// TwinCAT 3 PLC project ClientSampleProject
// ProgramVersion: 3.1.0.8
// libraries:
//   Tc2_Standard, * (Beckhoff Automation GmbH)
//   Tc2_System, * (Beckhoff Automation GmbH)
//   Tc3_Interfaces, * (Beckhoff Automation GmbH)
//   Tc3_Module, * (Beckhoff Automation GmbH)
//   Tc3_PLCopen_OpcUa, * (Beckhoff Automation GmbH)
//   Tc2_Utilities,newest,Beckhoff Automation GmbH
// project tree:
//   DUTs/ ST_OutputArgInfoAndData.TcDUT, ST_ReadListData.TcDUT (not stored), ST_ReadListData_Array.TcDUT
//   GVLs/ GlobalSettings.TcGVL
//   / PlcTask.TcTTO (not stored)
//   POUs/ MAIN.TcPOU, PRG_METHOD.TcPOU, PRG_READ.TcPOU, PRG_READ_IndexRange.TcPOU, PRG_READ_List.TcPOU, PRG_READ_List_Array.TcPOU, PRG_WRITE.TcPOU, PRG_WRITE_IndexRange.TcPOU
// (motion and I/O tree: see PLC project serversampleproject)
// real-time tasks:
//   TASK PlcTask: cycle T#10ms, priority 20, ADS port 350

// ---- DUTs/ST_OutputArgInfoAndData.TcDUT
{attribute 'pack_mode' := '1'}
TYPE ST_OutputArgInfoAndData :
STRUCT
	nNumberOfOutputArguments: UDINT; // determined amount of output parameters
	nReserved: ARRAY[1..4] OF BYTE; // Reserved padding
	stOutputArgInfo: ARRAY[1..1] OF ST_UAMethodArgInfo; // number of output parameters - M_Mul has 1 output parameter 
	pro: DINT;
END_STRUCT
END_TYPE

// ---- DUTs/ST_ReadListData_Array.TcDUT
{attribute 'pack_mode' := '1'}
TYPE ST_ReadListData_Array :
STRUCT
	stReadListReturnInfo	: ARRAY [1..2] OF ST_UAReadListReturnInfo;
	iArrayIntVar1 			: ARRAY[0..9] OF INT;
	iArrayIntVar2 			: ARRAY[0..11] OF INT;
END_STRUCT
END_TYPE

// ---- GVLs/GlobalSettings.TcGVL
VAR_GLOBAL
	(* These global connection and namespace settings need to be adapted to the runtime environment *)
	(*sOpcUaServerUrl : STRING(MAX_STRING_LENGTH) := 'opc.tcp://localhost:4840';
	sNamespaceUri : STRING(MAX_STRING_LENGTH) := 'urn:BeckhoffAutomation:Ua:PLC1'; // TF6100 setup version 4.x default*)
	
	sOpcUaServerUrl : STRING(MAX_STRING_LENGTH) := 'opc.tcp://172.17.36.240:4840';
	sNamespaceUri : STRING(MAX_STRING_LENGTH) := 'urn:BeckhoffAutomation:Ua:PLC1'; // TF6100 setup version 4.x default
END_VAR

// ---- POUs/MAIN.TcPOU
PROGRAM MAIN
VAR
	fbGetHostname : FB_GetHostName;
END_VAR

PRG_READ(); // Call sample for UA_Read
//PRG_READ_IndexRange(); // Call sample for UA_Read
//PRG_READ_List(); // Call sample for UA_ReadList
//PRG_READ_List_Array(); // Call sample for UA_ReadList to read array elements
//PRG_WRITE(); // Call sample for UA_Write
//PRG_WRITE_IndexRange(); // Call sample for UA_Write
//PRG_METHOD(); // Call sample for UA_MethodCall

END_PROGRAM

// ---- POUs/PRG_READ.TcPOU
PROGRAM PRG_READ
VAR
	(* Declarations for UA_Connect *)
	fbUA_Connect			: UA_Connect;
	SessionConnectInfo		: ST_UASessionConnectInfo;
	nConnectionHdl			: DWORD;

	(* Declarations for UA_GetNamespaceIndex *)
	fbUA_GetNamespaceIndex 	: UA_GetNamespaceIndex;
	nNamespaceIndex			: UINT;

	(* Declarations for UA_NodeGetHandle *)
	fbUA_NodeGetHandle		: UA_NodeGetHandle;
	NodeID					: ST_UANodeID;
	nNodeHdl				: DWORD;

	(* Declarations for UA_Read *)
	fbUA_Read				: UA_Read;
	stIndexRange			: ARRAY [1..nMaxIndexRange] OF ST_UAIndexRange;
	nIndexRangeCount		: UINT;
	stNodeAddInfo			: ST_UANodeAdditionalInfo;
	sNodeIdentifier			: STRING(MAX_STRING_LENGTH) := 'MAIN.nCounter'; // change to node identifier
	nReadData				: INT; 		// change to node data type
	cbDataRead				: UDINT;
	
	(* Declarations for UA_NodeReleaseHandle *)
	fbUA_NodeReleaseHandle	: UA_NodeReleaseHandle;

	(* Declarations for UA_Disconnect *)
	fbUA_Disconnect		: UA_Disconnect;

	(* Other declarations *)
	iState		: INT;
	bTest		: BOOL:= TRUE;
	bDone		: BOOL;
	bBusy		: BOOL;
	bError		: BOOL;
	nErrorID	: DWORD;
END_VAR


CASE iState OF
0:	(* idle *)
	IF bTest THEN
		bTest		:= FALSE;
		bError		:= FALSE;
		nErrorID	:= 0;

		SessionConnectInfo.tConnectTimeout 		:= T#1M;
		SessionConnectInfo.tSessionTimeout 		:= T#1M;
		SessionConnectInfo.sApplicationName		:= '';
		SessionConnectInfo.eSecurityMode 		:= eUASecurityMsgMode_Sign_Encrypt;
		SessionConnectInfo.eSecurityPolicyUri 	:= 5;
		SessionConnectInfo.eTransportProfileUri := eUATransportProfileUri_UATcp;

(*		nIndexRange[1].nStartIndex := 0;
		nIndexRange[1].nEndIndex := 1;
		nIndexRange[1].bRangeAccess := TRUE; *)
		stNodeAddInfo.nIndexRangeCount := nIndexRangeCount;
		stNodeAddInfo.stIndexRange := stIndexRange;
		iState	:= iState + 1;
	END_IF

1:	(* Open UA session *)
	fbUA_Connect(
		Execute				:= TRUE,
		ServerURL			:= sOpcUaServerUrl,
		SessionConnectInfo	:= SessionConnectInfo,
		Timeout				:= T#2M,
		ConnectionHdl		=> nConnectionHdl
	);

	IF NOT fbUA_Connect.Busy THEN
		fbUA_Connect(Execute := FALSE);

		IF NOT fbUA_Connect.Error THEN
			(* session open *)
			iState := iState + 1;
		ELSE
			bError			:= TRUE;
			nErrorID		:= fbUA_Connect.ErrorID;
			nConnectionHdl	:= 0;
			iState 			:= 0; (* idle *)
		END_IF
	END_IF


2:	(* GetNS Index *)
	fbUA_GetNamespaceIndex(
		Execute			:= TRUE,
		ConnectionHdl	:= nConnectionHdl,
		NamespaceUri	:= sNamespaceUri,
		NamespaceIndex	=> nNamespaceIndex
	);

	IF NOT fbUA_GetNamespaceIndex.Busy THEN
		fbUA_GetNamespaceIndex(Execute := FALSE);
		IF NOT fbUA_GetNamespaceIndex.Error THEN
			iState 		:= iState + 1;
		ELSE
			bError		:= TRUE;
			nErrorID	:= fbUA_GetNamespaceIndex.ErrorID;
			iState 		:= 6; (* idle *)
		END_IF
	END_IF

3:	(* Get Node Handle *)
	NodeID.eIdentifierType := eUAIdentifierType_String;
	NodeID.nNamespaceIndex := nNamespaceIndex;
	NodeID.sIdentifier	:= sNodeIdentifier;
	fbUA_NodeGetHandle(
		Execute			:= TRUE,
		ConnectionHdl	:= nConnectionHdl,
		NodeID			:= NodeID,
		NodeHdl			=> nNodeHdl
	);

	IF NOT fbUA_NodeGetHandle.Busy THEN
		fbUA_NodeGetHandle(Execute := FALSE);

		IF NOT fbUA_NodeGetHandle.Error THEN
			iState 		:= iState + 1;
		ELSE
			bError		:= TRUE;
			nErrorID	:= fbUA_NodeGetHandle.ErrorID;
			iState 		:= 6; (* idle *)
		END_IF
	END_IF


4: 	(* UA_Read *)
	fbUA_Read(
		Execute			:= TRUE,
		ConnectionHdl	:= nConnectionHdl,
		NodeHdl			:= nNodeHdl,
		cbData			:= SIZEOF(nReadData),
		stNodeAddInfo 	:= stNodeAddInfo,
		pVariable		:= ADR(nReadData)
		);

	IF NOT fbUA_Read.Busy THEN
		fbUA_Read( Execute := FALSE, cbData_R => cbDataRead);

		IF NOT fbUA_Read.Error THEN
			iState 		:= iState + 1;
		ELSE
			bError		:= TRUE;
			nErrorID	:= fbUA_Read.ErrorID;
			iState 		:= 6; (* idle *)
		END_IF
	END_IF


5:	(* Release Node Handle *)
	fbUA_NodeReleaseHandle(
		Execute			:= TRUE,
		ConnectionHdl	:= nConnectionHdl,
		NodeHdl			:= nNodeHdl
	);

	IF NOT fbUA_NodeReleaseHandle.Busy THEN
		fbUA_NodeReleaseHandle(Execute := FALSE);

		IF NOT fbUA_NodeReleaseHandle.Error THEN
			iState 		:= iState + 1;
		ELSE
			bError		:= TRUE;
			nErrorID	:= fbUA_NodeReleaseHandle.ErrorID;
			iState 		:= 6; (* idle *)
		END_IF
	END_IF


6:	(* close session *)
	fbUA_Disconnect(
		Execute			:= TRUE,
		ConnectionHdl	:= nConnectionHdl
	);

	IF NOT fbUA_Disconnect.Busy THEN
		fbUA_Disconnect(Execute := FALSE);
		bBusy := FALSE;
		IF NOT fbUA_Disconnect.Error THEN
			(* session closed *)
			iState 		:= 0;
			IF NOT bError THEN 
				bDone 	:= TRUE;
			END_IF
		ELSE
			bError			:= TRUE;
			nErrorID		:= fbUA_Disconnect.ErrorID;
			iState 			:= 0; (* idle *)
			nConnectionHdl	:= 0;
		END_IF
	END_IF
END_CASE

END_PROGRAM

// ---- POUs/PRG_METHOD.TcPOU
PROGRAM PRG_METHOD
VAR
	(* Declarations for UA_Connect *)	
	fbUA_Connect: UA_Connect;
	SessionConnectInfo: ST_UASessionConnectInfo;
	nConnectionHdl: DWORD;
	
	(* Declarations for UA_GetNamespaceIndex *)
	fbUA_GetNamespaceIndex: UA_GetNamespaceIndex;
	nNamespaceIndex: UINT;
	
	(* Declarations for UA_MethodGetHandle *)
	fbUA_MethodGetHandle: UA_MethodGetHandle;
	ObjectNodeID: ST_UANodeID;
	MethodNodeID: ST_UANodeID;
	nMethodHdl: DWORD;
	
	(* Declarations for UA_MethodCall *)
	fbUA_MethodCall: UA_MethodCall;
	sObjectNodeIdIdentifier	: STRING(MAX_STRING_LENGTH) := 'MAIN.fbMathematics'; // change to object node identifier (UAObject above method)
	sMethodNodeIdIdentifier : STRING(MAX_STRING_LENGTH) := 'MAIN.fbMathematics#M_Mul'; // change to method node identifier (UAMethod to call)
	nAdrWriteData: PVOID;
	numberIn1: INT := 42; // change according to input value and data type
	numberIn2: INT := 42; // change according to input value and data type
	numberOutPro: DINT; // result (output parameter of M_Mul())
	cbWriteData: UDINT; // calculated automatically by M_Init()
	InputArguments: ARRAY[1..2] OF ST_UAMethodArgInfo; // change according to input parameters - M_Mul has 2 input parameters 
	stOutputArgInfo: ARRAY[1..1] OF ST_UAMethodArgInfo; // change according to output parameters - M_Mul has 1 output parameters
	stOutputArgInfoAndData: ST_OutputArgInfoAndData;
	nInputData: ARRAY[1..4] OF BYTE; // numberIn1(INT16)(2) + numberIn2(INT16)(2)
	nOffset: UDINT; // calculated by M_Init()
	nArg: INT; // used by M_Init()
	
	(* Declarations for UA_MethodReleaseHandle *)
	fbUA_MethodReleaseHandle: UA_MethodReleaseHandle;

	(* Declarations for UA_Disconnect *)
	fbUA_Disconnect: UA_Disconnect;
			
	(* Other Declarations *)
	bTest: BOOL := TRUE;
	bDone: BOOL;
	bBusy: BOOL;
	bError: BOOL;
	nErrorID: DWORD;
	iState: INT;
	RTrig: R_TRIG;
	bInputDataError: BOOL;
END_VAR
VAR CONSTANT
	nInputArgSize: INT := 4; // numberIn1(INT16)(2) + numberIn2(INT16)(2)
	nNumberOfInputArguments: DINT := 2; // change to number of input parameters - M_Mul has 2 input parameters
	nNumberOfOutputArguments: DINT := 1; // change to number of output parameters - M_Mul has 1 output parameters
END_VAR

CASE iState OF

0:	(* idle *)
	IF bTest THEN
		bTest		:= FALSE;
		bError		:= FALSE;
		nErrorID	:= 0;

		SessionConnectInfo.tConnectTimeout 		:= T#1M;
		SessionConnectInfo.tSessionTimeout 		:= T#1M;
		SessionConnectInfo.sApplicationName		:= '';
		SessionConnectInfo.eSecurityMode 		:= eUASecurityMsgMode_None;
		SessionConnectInfo.eSecurityPolicyUri 	:= eUASecurityPolicy_None;
		SessionConnectInfo.eTransportProfileUri := eUATransportProfileUri_UATcp;

		iState	:= iState + 1;
	END_IF

	
1:	(* open UA session *)
	fbUA_Connect(
		Execute				:= TRUE,
		ServerURL			:= sOpcUaServerUrl,
		SessionConnectInfo	:= SessionConnectInfo,
		Timeout				:= T#2M,
		ConnectionHdl		=> nConnectionHdl
	);

	IF NOT fbUA_Connect.Busy THEN
		fbUA_Connect(Execute := FALSE);

		IF NOT fbUA_Connect.Error THEN
			(* connected *)
			iState := iState + 1;
		ELSE
			bError			:= TRUE;
			nErrorID		:= fbUA_Connect.ErrorID;
			nConnectionHdl	:= 0;
			iState 			:= 0; (* idle *)
		END_IF
	END_IF


2:	(* GetNS Index *)
	fbUA_GetNamespaceIndex(
		Execute			:= TRUE,
		ConnectionHdl	:= nConnectionHdl,
		NamespaceUri	:= sNamespaceUri,
		NamespaceIndex	=> nNamespaceIndex
	);

	IF NOT fbUA_GetNamespaceIndex.Busy THEN
		fbUA_GetNamespaceIndex(Execute := FALSE);

		IF NOT fbUA_GetNamespaceIndex.Error THEN
			(* namespace index read successfully *)
			iState 		:= iState + 1;
		ELSE
			bError		:= TRUE;
			nErrorID	:= fbUA_GetNamespaceIndex.ErrorID;
			iState 		:= 7; (* disconnect *)
		END_IF
	END_IF

	
3:	(* Get Method Handle *)
	ObjectNodeID.eIdentifierType := eUAIdentifierType_String;
	ObjectNodeID.nNamespaceIndex := nNamespaceIndex;
	ObjectNodeID.sIdentifier	 := sObjectNodeIdIdentifier;

	MethodNodeID.eIdentifierType := eUAIdentifierType_String;
	MethodNodeID.nNamespaceIndex := nNamespaceIndex;
	MethodNodeID.sIdentifier	 := sMethodNodeIdIdentifier;

	M_Init();
	IF bInputDataError = FALSE THEN
		iState 	:= iState + 1;
	ELSE
		bBusy		:= FALSE;  
		bError 		:= TRUE;
		nErrorID 	:= 16#70A; //out of memory
	END_IF

	
4:	(* Method Get Handle *)
	fbUA_MethodGetHandle(
			Execute			:= TRUE,
			ConnectionHdl	:= nConnectionHdl,
			ObjectNodeID	:= ObjectNodeID,
			MethodNodeID 	:= MethodNodeID,
			MethodHdl		=> nMethodHdl
		);
	IF NOT fbUA_MethodGetHandle.Busy THEN
		fbUA_MethodGetHandle(Execute := FALSE);

		IF NOT fbUA_MethodGetHandle.Error THEN
			(*  *)
			iState := iState + 1; (* Call Method *)
		ELSE
			bError		:= TRUE;
			nErrorID	:= fbUA_MethodGetHandle.ErrorID;
			iState	 	:= 6; (* Release method Handle *)
		END_IF
	END_IF


5:	(* Method Call *)
	stOutputArgInfo[1].nLenData := SIZEOF(stOutputArgInfoAndData.pro);
	fbUA_MethodCall(
		Execute					:= TRUE,
		ConnectionHdl			:= nConnectionHdl,
		MethodHdl				:= nMethodHdl,
		nNumberOfInputArguments := nNumberOfInputArguments,	
		pInputArgInfo			:= ADR(InputArguments),
		cbInputArgInfo			:= SIZEOF(InputArguments),
		pInputArgData			:= ADR(nInputData),
		cbInputArgData			:= cbWriteData,
		pInputWriteData			:= 0,
		cbInputWriteData		:= 0,
		nNumberOfOutputArguments:= nNumberOfOutputArguments,
		pOutputArgInfo			:= ADR(stOutputArgInfo),
		cbOutputArgInfo			:= SIZEOF(stOutputArgInfo),
		pOutputArgInfoAndData	:= ADR(stOutputArgInfoAndData),
		cbOutputArgInfoAndData	:= SIZEOF(stOutputArgInfoAndData),		
	);
	IF NOT fbUA_MethodCall.Busy THEN
		fbUA_MethodCall(Execute := FALSE);
		IF NOT fbUA_MethodCall.Error THEN
			(* clear data and restart *)
			iState := iState + 1; (* Release handle *)
			numberOutPro := stOutputArgInfoAndData.pro;
		ELSE
			bError		:= TRUE;
			nErrorID	:= fbUA_MethodCall.ErrorID;
			iState		:= 6; (* Release method handle *)
		END_IF
	END_IF


6:	(* Release Method Handle *)
	fbUA_MethodReleaseHandle(
		Execute			:= TRUE,
		ConnectionHdl	:= nConnectionHdl,
		MethodHdl		:= nMethodHdl
	);

	IF NOT fbUA_MethodReleaseHandle.Busy THEN
		fbUA_MethodReleaseHandle(Execute := FALSE);
		bBusy := FALSE;
		IF NOT fbUA_MethodReleaseHandle.Error THEN
			(* session closed *)
			iState 	:= 7; (* Disconnect *)
		ELSE
			bError		:= TRUE;
			nErrorID	:= fbUA_MethodReleaseHandle.ErrorID;
			iState 		:= 7; (* Disconnect *)
		END_IF
	END_IF
	
	
7:	(* Disconnect *) 
	fbUA_Disconnect(
		Execute			:= TRUE,
		ConnectionHdl	:= nConnectionHdl
	);

	IF NOT fbUA_Disconnect.Busy THEN
		fbUA_Disconnect(Execute := FALSE);

		IF NOT fbUA_Disconnect.Error THEN
			(* disconnected *)
			iState 	:= 0; (* idle *)
			bDone 	:= TRUE;
			bBusy 	:= FALSE;
		ELSE
			bBusy 			:= FALSE;
			bError			:= TRUE;
			nErrorID		:= fbUA_Disconnect.ErrorID;
			iState 			:= 0; (* idle *)
			nConnectionHdl	:= 0;
		END_IF
	END_IF
END_CASE

ACTION M_Init:
bInputDataError := FALSE; 
nOffset := 0;
MEMSET(ADR(InputArguments),0,SIZEOF(InputArguments));
MEMSET(ADR(nInputData),0,SIZEOF(nInputData));

nArg := 1;
(*numberIn1*)			(********** Input parameter 1 **********)
InputArguments[nArg].DataType			:= eUAType_Int16;
InputArguments[nArg].ValueRank			:= -1; 							(* Scalar = -1 or Array *)
InputArguments[nArg].ArrayDimensions[1]	:= 0; 							(* Number of Dimension in case its an array *)
InputArguments[nArg].nLenData			:= SIZEOF(numberIn1);			(* Length if its a STRING *)
IF nOffset + SIZEOF(numberIn1) > nInputArgSize THEN 
	bInputDataError := TRUE;
	RETURN;
ELSE
	MEMCPY(ADR(nInputData)+nOffset,ADR(numberIn1),SIZEOF(numberIn1));				(* VALUE in BYTES FORM *)
	nOffset := nOffset + SIZEOF(numberIn1);
END_IF

nArg := nArg + 1;
(* numberIn2;*)			(********** Input parameter 2 **********)
InputArguments[nArg].DataType			:= eUAType_Int16;
InputArguments[nArg].ValueRank			:= -1; 							(* Scalar = -1 or Array *)
InputArguments[nArg].ArrayDimensions[1]	:= 0; 							(* Number of Dimension in case its an array *)
InputArguments[nArg].nLenData			:= SIZEOF(numberIn2);				(* Length if its a STRING *)
IF nOffset + SIZEOF(numberIn2) > nInputArgSize THEN 
	bInputDataError := TRUE;
	RETURN;
ELSE
	MEMCPY(ADR(nInputData)+nOffset,ADR(numberIn2),SIZEOF(numberIn2));			(* VALUE in BYTES FORM *)
	nOffset := nOffset + SIZEOF(numberIn2);
END_IF

cbWriteData := nOffset;
END_ACTION

END_PROGRAM

// ---- POUs/PRG_READ_IndexRange.TcPOU
PROGRAM PRG_READ_IndexRange
VAR
	(* Declarations for UA_Connect *)
	fbUA_Connect			: UA_Connect;
	SessionConnectInfo		: ST_UASessionConnectInfo;
	nConnectionHdl			: DWORD;

	(* Declarations for UA_GetNamespaceIndex *)
	fbUA_GetNamespaceIndex 	: UA_GetNamespaceIndex;
	nNamespaceIndex			: UINT;

	(* Declarations for UA_NodeGetHandle *)
	fbUA_NodeGetHandle		: UA_NodeGetHandle;
	NodeID					: ST_UANodeID;
	nNodeHdl				: DWORD;

	(* Declarations for UA_Read *)
	fbUA_Read				: UA_Read;
	stIndexRange			: ARRAY [1..nMaxIndexRange] OF ST_UAIndexRange;
	//nIndexRangeCount		: UINT;
	stNodeAddInfo			: ST_UANodeAdditionalInfo;
	sNodeIdentifier			: STRING(MAX_STRING_LENGTH) := 'MAIN.iArrayIntVar3'; // change to node identifier
	nReadData				: ARRAY[0..3] OF DINT; 		// change to node data type
	cbDataRead				: UDINT;
	
	(* Declarations for UA_NodeReleaseHandle *)
	fbUA_NodeReleaseHandle	: UA_NodeReleaseHandle;

	(* Declarations for UA_Disconnect *)
	fbUA_Disconnect		: UA_Disconnect;

	(* Other declarations *)
	iState		: INT;
	bTest		: BOOL:= TRUE;
	bDone		: BOOL;
	bBusy		: BOOL;
	bError		: BOOL;
	nErrorID	: DWORD;
END_VAR


CASE iState OF
0:	(* idle *)
	IF bTest THEN
		bTest		:= FALSE;
		bError		:= FALSE;
		nErrorID	:= 0;

		SessionConnectInfo.tConnectTimeout 		:= T#1M;
		SessionConnectInfo.tSessionTimeout 		:= T#1M;
		SessionConnectInfo.sApplicationName		:= '';
		SessionConnectInfo.eSecurityMode 		:= eUASecurityMsgMode_None;
		SessionConnectInfo.eSecurityPolicyUri 	:= eUASecurityPolicy_None;
		SessionConnectInfo.eTransportProfileUri := eUATransportProfileUri_UATcp;

		stIndexRange[1].nStartIndex := 2;
		stIndexRange[1].nEndIndex := 5;
		stNodeAddInfo.nIndexRangeCount := 1;
		stNodeAddInfo.stIndexRange := stIndexRange;
		
		iState	:= iState + 1;
	END_IF

1:	(* Open UA session *)
	fbUA_Connect(
		Execute				:= TRUE,
		ServerURL			:= sOpcUaServerUrl,
		SessionConnectInfo	:= SessionConnectInfo,
		Timeout				:= T#2M,
		ConnectionHdl		=> nConnectionHdl
	);

	IF NOT fbUA_Connect.Busy THEN
		fbUA_Connect(Execute := FALSE);

		IF NOT fbUA_Connect.Error THEN
			(* session open *)
			iState := iState + 1;
		ELSE
			bError			:= TRUE;
			nErrorID		:= fbUA_Connect.ErrorID;
			nConnectionHdl	:= 0;
			iState 			:= 0; (* idle *)
		END_IF
	END_IF


2:	(* GetNS Index *)
	fbUA_GetNamespaceIndex(
		Execute			:= TRUE,
		ConnectionHdl	:= nConnectionHdl,
		NamespaceUri	:= sNamespaceUri,
		NamespaceIndex	=> nNamespaceIndex
	);

	IF NOT fbUA_GetNamespaceIndex.Busy THEN
		fbUA_GetNamespaceIndex(Execute := FALSE);
		IF NOT fbUA_GetNamespaceIndex.Error THEN
			iState 		:= iState + 1;
		ELSE
			bError		:= TRUE;
			nErrorID	:= fbUA_GetNamespaceIndex.ErrorID;
			iState 		:= 6; (* idle *)
		END_IF
	END_IF

3:	(* Get Node Handle *)
	NodeID.eIdentifierType := eUAIdentifierType_String;
	NodeID.nNamespaceIndex := nNamespaceIndex;
	NodeID.sIdentifier	:= sNodeIdentifier;
	fbUA_NodeGetHandle(
		Execute			:= TRUE,
		ConnectionHdl	:= nConnectionHdl,
		NodeID			:= NodeID,
		NodeHdl			=> nNodeHdl
	);

	IF NOT fbUA_NodeGetHandle.Busy THEN
		fbUA_NodeGetHandle(Execute := FALSE);

		IF NOT fbUA_NodeGetHandle.Error THEN
			iState 		:= iState + 1;
		ELSE
			bError		:= TRUE;
			nErrorID	:= fbUA_NodeGetHandle.ErrorID;
			iState 		:= 6; (* idle *)
		END_IF
	END_IF


4: 	(* UA_Read *)
	fbUA_Read(
		Execute			:= TRUE,
		ConnectionHdl	:= nConnectionHdl,
		NodeHdl			:= nNodeHdl,
		cbData			:= SIZEOF(nReadData),
		stNodeAddInfo 	:= stNodeAddInfo,
		pVariable		:= ADR(nReadData)
		);

	IF NOT fbUA_Read.Busy THEN
		fbUA_Read( Execute := FALSE, cbData_R => cbDataRead);

		IF NOT fbUA_Read.Error THEN
			iState 		:= iState + 1;
		ELSE
			bError		:= TRUE;
			nErrorID	:= fbUA_Read.ErrorID;
			iState 		:= 6; (* idle *)
		END_IF
	END_IF


5:	(* Release Node Handle *)
	fbUA_NodeReleaseHandle(
		Execute			:= TRUE,
		ConnectionHdl	:= nConnectionHdl,
		NodeHdl			:= nNodeHdl
	);

	IF NOT fbUA_NodeReleaseHandle.Busy THEN
		fbUA_NodeReleaseHandle(Execute := FALSE);

		IF NOT fbUA_NodeReleaseHandle.Error THEN
			iState 		:= iState + 1;
		ELSE
			bError		:= TRUE;
			nErrorID	:= fbUA_NodeReleaseHandle.ErrorID;
			iState 		:= 6; (* idle *)
		END_IF
	END_IF


6:	(* close session *)
	fbUA_Disconnect(
		Execute			:= TRUE,
		ConnectionHdl	:= nConnectionHdl
	);

	IF NOT fbUA_Disconnect.Busy THEN
		fbUA_Disconnect(Execute := FALSE);
		bBusy := FALSE;
		IF NOT fbUA_Disconnect.Error THEN
			(* session closed *)
			iState 		:= 0;
			IF NOT bError THEN 
				bDone 	:= TRUE;
			END_IF
		ELSE
			bError			:= TRUE;
			nErrorID		:= fbUA_Disconnect.ErrorID;
			iState 			:= 0; (* idle *)
			nConnectionHdl	:= 0;
		END_IF
	END_IF
END_CASE

END_PROGRAM

// ---- POUs/PRG_READ_List.TcPOU
PROGRAM PRG_READ_List
VAR
	fbUA_ConnectEx			: UA_Connect;
	SessionConnectInfoEx	: ST_UASessionConnectInfo;
	sOpcUA_URL				: STRING(MAX_STRING_LENGTH);
	nConnectionHdl			: DWORD;

	fbUA_GetNamespaceIndex 	: UA_GetNamespaceIndex;
	nNamespaceIndex			: UINT;
	fbUA_NodeGetHandleList	: UA_NodeGetHandleList;
	
	NodeIDs					: ARRAY [1..nMaxNodeIDsInList] OF ST_UANodeID;
	nNodeHdls				: ARRAY [1..nMaxNodeIDsInList] OF DWORD;

	fbUA_ReadList			: UA_ReadList;
	NodeIDCount				: UINT := 2;
	NodeHdlCount			: UINT := 2; 
	stIndexRange			: ARRAY [1..nMaxIndexRange] OF ST_UAIndexRange;
	nIndexRangeCount		: UINT;
	stNodeAddInfo			: ARRAY [1..nMaxNodeIDsInList] OF ST_UANodeAdditionalInfo;
	stReadListData			: ST_ReadListData; // memory block must contain the Data[], NodeErrorIDs[], TimeStamps[] and cbData_R[]
	cbData					: ARRAY [1..nMaxNodeIDsInList] OF UDINT; (* Bytes to be actually Read *)
	cbData_R				: UDINT;
	cbDataTotal				: UDINT; 
	
	fbUA_NodeReleaseHandleList	: UA_NodeReleaseHandleList;

	fbUA_Disconnect		: UA_Disconnect;

	iState		: INT;
	bTest		: BOOL:= TRUE;
	bDone		: BOOL;
	bBusy		: BOOL;
	bError		: BOOL;
	nErrorID	: DWORD;
END_VAR


CASE iState OF
0:	(* idle *)
	IF bTest THEN
		bTest		:= FALSE;
		bError		:= FALSE;
		nErrorID	:= 0;

		SessionConnectInfoEx.tConnectTimeout 		:= T#1M;
		SessionConnectInfoEx.tSessionTimeout 		:= T#1M;
		SessionConnectInfoEx.sApplicationName		:= '';
		SessionConnectInfoEx.eSecurityMode 			:= eUASecurityMsgMode_None;
		SessionConnectInfoEx.eSecurityPolicyUri 	:= eUASecurityPolicy_None;
		SessionConnectInfoEx.eTransportProfileUri 	:= eUATransportProfileUri_UATcp;

		iState	:= iState + 1;
	END_IF

1:	(* open UA session *)
	fbUA_ConnectEx(
		Execute				:= TRUE,
		ServerURL			:= sOpcUaServerUrl,
		SessionConnectInfo  := SessionConnectInfoEx,
		Timeout				:= T#2M,
		ConnectionHdl		=> nConnectionHdl
	);

	IF NOT fbUA_ConnectEx.Busy THEN
		fbUA_ConnectEx(Execute := FALSE);

		IF NOT fbUA_ConnectEx.Error THEN
			(* session open *)
			iState := iState + 1;
		ELSE
			bError			:= TRUE;
			nErrorID		:= fbUA_ConnectEx.ErrorID;
			nConnectionHdl	:= 0;
			iState 			:= 0; (* idle *)
		END_IF
	END_IF


2:	(* GetNS Index *)
	fbUA_GetNamespaceIndex(
		Execute			:= TRUE,
		ConnectionHdl	:= nConnectionHdl,
		NamespaceUri	:= sNamespaceUri,
		NamespaceIndex	=> nNamespaceIndex
	);

	IF NOT fbUA_GetNamespaceIndex.Busy THEN
		fbUA_GetNamespaceIndex(Execute := FALSE);
		IF NOT fbUA_GetNamespaceIndex.Error THEN
			(* session closed *)
			iState 		:= iState + 1; (* idle *)
		ELSE
			bError		:= TRUE;
			nErrorID	:= fbUA_GetNamespaceIndex.ErrorID;
			iState 		:= 6; (* idle *)
		END_IF
	END_IF


3:	(* Get Node Handle *)
	
	NodeIDs[1].eIdentifierType := eUAIdentifierType_String;
	NodeIDs[1].nNamespaceIndex := nNamespaceIndex;
	NodeIDs[1].sIdentifier	:= 'MAIN.iVar1';
	
	NodeIDs[2].eIdentifierType := eUAIdentifierType_String;
	NodeIDs[2].nNamespaceIndex := nNamespaceIndex;
	NodeIDs[2].sIdentifier	:= 'MAIN.iVar2';

	fbUA_NodeGetHandleList(
		Execute			:= TRUE,
		ConnectionHdl	:= nConnectionHdl,
		NodeIDCount 	:= NodeIDCount,
		NodeIDs			:= NodeIDs,
		NodeHdls		=> nNodeHdls
	);

	IF NOT fbUA_NodeGetHandleList.Busy THEN
		fbUA_NodeGetHandleList(Execute := FALSE);

		IF NOT fbUA_NodeGetHandleList.Error THEN
			(* session closed *)
			iState 		:= iState + 1; (* idle *)
		ELSE
			bError		:= TRUE;
			nErrorID	:= fbUA_NodeGetHandleList.ErrorID;
			iState 		:= 6; (* idle *)
		END_IF
	END_IF

	
4: 	(* UA_Read *)
	cbData[1] := SIZEOF(stReadListData.nIntVar1);
	cbData[2] := SIZEOF(stReadListData.nIntVar2);
	cbDataTotal := SIZEOF(stReadListData);
	fbUA_ReadList(
		Execute			:= TRUE,
		ConnectionHdl	:= nConnectionHdl,
		NodeHdlCount	:= NodeHdlCount, // 2
		NodeHdls		:= nNodeHdls,
		stNodeAddInfo 	:= stNodeAddInfo,
		pVariable		:= ADR(stReadListData),
		cbData			:= cbData ,
		cbDataTotal		:= cbDataTotal		
		);

	IF NOT fbUA_ReadList.Busy THEN
		fbUA_ReadList( Execute := FALSE, cbData_R => cbData_R);

		IF NOT fbUA_ReadList.Error THEN
			(* session closed *)
			iState 		:= iState + 1; (* idle *)
		ELSE
			bError		:= TRUE;
			nErrorID	:= fbUA_ReadList.ErrorID;
			iState 		:= 6; (* idle *)
		END_IF
	END_IF


5:	(* Release Node Handle *)
	fbUA_NodeReleaseHandleList(
		Execute			:= TRUE,
		ConnectionHdl	:= nConnectionHdl,
		NodeHdlCount	:= NodeHdlCount,
		NodeHdls		:= nNodeHdls
	);

	IF NOT fbUA_NodeReleaseHandleList.Busy THEN
		fbUA_NodeReleaseHandleList(Execute := FALSE);

		IF NOT fbUA_NodeReleaseHandleList.Error THEN
			(* session closed *)
			iState 		:= iState + 1; (* idle *)
		ELSE
			bError		:= TRUE;
			nErrorID	:= fbUA_NodeReleaseHandleList.ErrorID;
			iState 		:= 6; (* idle *)
		END_IF
	END_IF


6:	(* close session *)
	fbUA_Disconnect(
		Execute			:= TRUE,
		ConnectionHdl	:= nConnectionHdl
	);

	IF NOT fbUA_Disconnect.Busy THEN
		fbUA_Disconnect(Execute := FALSE);
		bBusy := FALSE;
		IF NOT fbUA_Disconnect.Error THEN
			(* session closed *)
			iState 		:= 0; (* idle *)
			IF NOT bError THEN 
				bDone 	:= TRUE;
			END_IF
		ELSE
			bError			:= TRUE;
			nErrorID		:= fbUA_Disconnect.ErrorID;
			iState 			:= 0; (* idle *)
			nConnectionHdl	:= 0;
		END_IF
	END_IF
END_CASE

END_PROGRAM

// ---- POUs/PRG_READ_List_Array.TcPOU
PROGRAM PRG_READ_List_Array
VAR
	fbUA_Connect			: UA_Connect;
	SessionConnectInfo		: ST_UASessionConnectInfo;
	sOpcUA_URL				: STRING(MAX_STRING_LENGTH);
	nConnectionHdl			: DWORD;

	fbUA_GetNamespaceIndex 	: UA_GetNamespaceIndex;
	nNamespaceIndex			: UINT;
	fbUA_NodeGetHandleList	: UA_NodeGetHandleList;
	NodeIDs					: ARRAY [1..nMaxNodeIDsInList] OF ST_UANodeID;
	nNodeHdls				: ARRAY [1..nMaxNodeIDsInList] OF DWORD;

	fbUA_ReadList			: UA_ReadList; 
	stIndexRange			: ARRAY [1..nMaxIndexRange] OF ST_UAIndexRange;
	nIndexRangeCount		: UINT;
	stNodeAddInfo			: ARRAY [1..nMaxNodeIDsInList] OF ST_UANodeAdditionalInfo;
	stReadListDataArrayInt	: ST_ReadListData_Array; // memory block must contain the Data[], NodeErrorIDs[], TimeStamps[] and cbData_R[]
	cbData					: ARRAY [1..nMaxNodeIDsInList] OF UDINT; (* Bytes to be actually Read *)
	cbData_R				: UDINT;
	cbDataTotal				: UDINT; 
	
	fbUA_NodeReleaseHandleList	: UA_NodeReleaseHandleList;

	fbUA_Disconnect		: UA_Disconnect;

	iState		: INT;
	bTest		: BOOL:= TRUE;
	bDone		: BOOL;
	bBusy		: BOOL;
	bError		: BOOL;
	nErrorID	: DWORD;
	
	nNodeIdx	: INT; 
END_VAR


CASE iState OF
0:	(* idle *)
	IF bTest THEN
		bTest		:= FALSE;
		bError		:= FALSE;
		nErrorID	:= 0;

		SessionConnectInfo.tConnectTimeout 		:= T#1M;
		SessionConnectInfo.tSessionTimeout 		:= T#1M;
		SessionConnectInfo.sApplicationName		:= '';
		SessionConnectInfo.eSecurityMode 		:= eUASecurityMsgMode_None;
		SessionConnectInfo.eSecurityPolicyUri 	:= eUASecurityPolicy_None;
		SessionConnectInfo.eTransportProfileUri := eUATransportProfileUri_UATcp;

		iState	:= iState + 1;
	END_IF

1:	(* open UA session *)
	fbUA_Connect(
		Execute				:= TRUE,
		ServerURL			:= sOpcUaServerUrl,
		SessionConnectInfo  := SessionConnectInfo,
		Timeout				:= T#2M,
		ConnectionHdl		=> nConnectionHdl
	);

	IF NOT fbUA_Connect.Busy THEN
		fbUA_Connect(Execute := FALSE);

		IF NOT fbUA_Connect.Error THEN
			(* session open *)
			iState := iState + 1;
		ELSE
			bError			:= TRUE;
			nErrorID		:= fbUA_Connect.ErrorID;
			nConnectionHdl	:= 0;
			iState 			:= 0; (* idle *)
		END_IF
	END_IF


2:	(* GetNS Index *)
	fbUA_GetNamespaceIndex(
		Execute			:= TRUE,
		ConnectionHdl	:= nConnectionHdl,
		NamespaceUri	:= sNamespaceUri,
		NamespaceIndex	=> nNamespaceIndex
	);

	IF NOT fbUA_GetNamespaceIndex.Busy THEN
		fbUA_GetNamespaceIndex(Execute := FALSE);
		IF NOT fbUA_GetNamespaceIndex.Error THEN
			(* session closed *)
			iState 		:= iState + 1; (* idle *)
		ELSE
			bError		:= TRUE;
			nErrorID	:= fbUA_GetNamespaceIndex.ErrorID;
			iState 		:= 6; (* idle *)
		END_IF
	END_IF


3:	(* Get Node Handle *)

	nNodeIdx := 1;
	NodeIDs[nNodeIdx].eIdentifierType := eUAIdentifierType_String;
	NodeIDs[nNodeIdx].nNamespaceIndex := nNamespaceIndex;
	NodeIDs[nNodeIdx].sIdentifier	:= 'MAIN.iArrayIntVar1';
	
	nNodeIdx := nNodeIdx + 1;
	NodeIDs[nNodeIdx].eIdentifierType := eUAIdentifierType_String;
	NodeIDs[nNodeIdx].nNamespaceIndex := nNamespaceIndex;
	NodeIDs[nNodeIdx].sIdentifier	:= 'MAIN.iArrayIntVar2';

	fbUA_NodeGetHandleList(
		Execute			:= TRUE,
		ConnectionHdl	:= nConnectionHdl,
		NodeIDCount 	:= nNodeIdx,
		NodeIDs			:= NodeIDs,
		NodeHdls		=> nNodeHdls
	);

	IF NOT fbUA_NodeGetHandleList.Busy THEN
		fbUA_NodeGetHandleList(Execute := FALSE);

		IF NOT fbUA_NodeGetHandleList.Error THEN
			(* session closed *)
			iState 		:= iState + 1; (* idle *)
		ELSE
			bError		:= TRUE;
			nErrorID	:= fbUA_NodeGetHandleList.ErrorID;
			iState 		:= 6; (* idle *)
		END_IF
	END_IF

	
4: 	(* UA_Read *)
	cbData[1] := SIZEOF(stReadListDataArrayInt.iArrayIntVar1);
	cbData[2] := SIZEOF(stReadListDataArrayInt.iArrayIntVar2);

	cbDataTotal := SIZEOF(stReadListDataArrayInt);
	fbUA_ReadList(
		Execute			:= TRUE,
		ConnectionHdl	:= nConnectionHdl,
		NodeHdlCount	:= nNodeIdx, // 2
		NodeHdls		:= nNodeHdls,
		stNodeAddInfo 	:= stNodeAddInfo,
		pVariable		:= ADR(stReadListDataArrayInt),
		cbData			:= cbData ,
		cbDataTotal		:= cbDataTotal		
		);

	IF NOT fbUA_ReadList.Busy THEN
		fbUA_ReadList( Execute := FALSE, cbData_R => cbData_R);

		IF NOT fbUA_ReadList.Error THEN
			(* session closed *)
			iState 		:= iState + 1; (* idle *)
		ELSE
			bError		:= TRUE;
			nErrorID	:= fbUA_ReadList.ErrorID;
			iState 		:= 6; (* idle *)
		END_IF
	END_IF


5:	(* Release Node Handle *)
	fbUA_NodeReleaseHandleList(
		Execute			:= TRUE,
		ConnectionHdl	:= nConnectionHdl,
		NodeHdlCount	:= nNodeIdx,
		NodeHdls		:= nNodeHdls
	);

	IF NOT fbUA_NodeReleaseHandleList.Busy THEN
		fbUA_NodeReleaseHandleList(Execute := FALSE);

		IF NOT fbUA_NodeReleaseHandleList.Error THEN
			(* session closed *)
			iState 		:= iState + 1; (* idle *)
		ELSE
			bError		:= TRUE;
			nErrorID	:= fbUA_NodeReleaseHandleList.ErrorID;
			iState 		:= 6; (* idle *)
		END_IF
	END_IF


6:	(* close session *)
	fbUA_Disconnect(
		Execute			:= TRUE,
		ConnectionHdl	:= nConnectionHdl
	);

	IF NOT fbUA_Disconnect.Busy THEN
		fbUA_Disconnect(Execute := FALSE);
		bBusy := FALSE;
		IF NOT fbUA_Disconnect.Error THEN
			(* session closed *)
			iState 		:= 0; (* idle *)
			IF NOT bError THEN 
				bDone 	:= TRUE;
			END_IF
		ELSE
			bError			:= TRUE;
			nErrorID		:= fbUA_Disconnect.ErrorID;
			iState 			:= 0; (* idle *)
			nConnectionHdl	:= 0;
		END_IF
	END_IF
END_CASE

END_PROGRAM

// ---- POUs/PRG_WRITE.TcPOU
PROGRAM PRG_WRITE
VAR
	(* Declarations for UA_Connect *)
	fbUA_Connect			: UA_Connect;
	SessionConnectInfo		: ST_UASessionConnectInfo;
	nConnectionHdl			: DWORD;

	(* Declarations for UA_GetNamespaceIndex *)
	fbUA_GetNamespaceIndex 	: UA_GetNamespaceIndex;
	nNamespaceIndex			: UINT;

	(* Declarations for UA_NodeGetHandle *)
	fbUA_NodeGetHandle		: UA_NodeGetHandle;
	NodeID					: ST_UANodeID;
	nNodeHdl				: DWORD;

	(* Declarations for UA_Write *)
	fbUA_Write				: UA_Write;
	stIndexRange			: ARRAY [1..nMaxIndexRange] OF ST_UAIndexRange;
	nIndexRangeCount		: UINT;
	stNodeAddInfo			: ST_UANodeAdditionalInfo;
	sNodeIdentifier			: STRING(MAX_STRING_LENGTH) := 'MAIN.nNumber'; // change to node identifier
	nWriteData				: INT := 42;		// change according to the type of variable that should be written
	
	(* Declarations for UA_NodeReleaseHandle *)
	fbUA_NodeReleaseHandle	: UA_NodeReleaseHandle;

	(* Declarations for UA_Disconnect *)
	fbUA_Disconnect			: UA_Disconnect;

	(* Other declarations *)
	iState			: INT;
	bTest			: BOOL := TRUE;
	bDone			: BOOL;
	bBusy			: BOOL;
	bError			: BOOL;
	nErrorID		: DWORD;
END_VAR

CASE iState OF
0:	(* idle *)
	IF bTest THEN
		bTest	:= FALSE;
		bError	:= FALSE;
		nErrorID	:= 0;

		SessionConnectInfo.tConnectTimeout 		:= T#1M;
		SessionConnectInfo.tSessionTimeout 		:= T#1M;
		SessionConnectInfo.sApplicationName		:= '';
		SessionConnectInfo.eSecurityMode 		:= eUASecurityMsgMode_None;
		SessionConnectInfo.eSecurityPolicyUri 	:= eUASecurityPolicy_None;
		SessionConnectInfo.eTransportProfileUri := eUATransportProfileUri_UATcp;

		stNodeAddInfo.nIndexRangeCount := nIndexRangeCount;
		stNodeAddInfo.stIndexRange := stIndexRange;
		iState	:= iState + 1;
	END_IF

1:	(* open UA session *)
	fbUA_Connect(
		Execute				:= TRUE,
		ServerURL			:= sOpcUaServerUrl,
		SessionConnectInfo	:= SessionConnectInfo,
		Timeout				:= T#2M,
		ConnectionHdl		=> nConnectionHdl
	);

	IF NOT fbUA_Connect.Busy THEN
		fbUA_Connect(Execute := FALSE);

		IF NOT fbUA_Connect.Error THEN
			(* session open *)
			iState := iState + 1;
		ELSE
			bError			:= TRUE;
			nErrorID		:= fbUA_Connect.ErrorID;
			nConnectionHdl	:= 0;
			iState 			:= 0; (* idle *)
		END_IF
	END_IF


2:	(* GetNS Index *)
	fbUA_GetNamespaceIndex(
		Execute			:= TRUE,
		ConnectionHdl	:= nConnectionHdl,
		NamespaceUri	:= sNamespaceUri,
		NamespaceIndex	=> nNamespaceIndex
	);

	IF NOT fbUA_GetNamespaceIndex.Busy THEN
		fbUA_GetNamespaceIndex(Execute := FALSE);

		IF NOT fbUA_GetNamespaceIndex.Error THEN
			iState 		:= iState + 1;
		ELSE
			bError		:= TRUE;
			nErrorID	:= fbUA_GetNamespaceIndex.ErrorID;
			iState 		:= 6; (* idle *)
		END_IF
	END_IF


3:	(* Get Node Handle *)
	NodeID.eIdentifierType := eUAIdentifierType_String;
	NodeID.nNamespaceIndex := nNamespaceIndex;
	NodeID.sIdentifier	:= sNodeIdentifier;
	fbUA_NodeGetHandle(
		Execute			:= TRUE,
		ConnectionHdl	:= nConnectionHdl,
		NodeID			:= NodeID,
		NodeHdl			=> nNodeHdl
	);

	IF NOT fbUA_NodeGetHandle.Busy THEN
		fbUA_NodeGetHandle(Execute := FALSE);

		IF NOT fbUA_NodeGetHandle.Error THEN
			iState 		:= iState + 1;
		ELSE
			bError		:= TRUE;
			nErrorID	:= fbUA_NodeGetHandle.ErrorID;
			iState 		:= 6; (* idle *)
		END_IF
	END_IF


4: 	(* UA_Write *)
	fbUA_Write(
		Execute			:= TRUE,
		ConnectionHdl	:= nConnectionHdl,
		NodeHdl			:= nNodeHdl,
		stNodeAddInfo	:= stNodeAddInfo,
		cbData			:= SIZEOF(nWriteData),
		pVariable		:= ADR(nWriteData)
		);

	IF NOT fbUA_Write.Busy THEN
		fbUA_Write(
			Execute 	:= FALSE,
			pVariable	:= ADR(nWriteData));

		IF NOT fbUA_Write.Error THEN
			iState 		:= iState + 1;
		ELSE
			bError		:= TRUE;
			nErrorID	:= fbUA_Write.ErrorID;
			iState 		:= 6; (* idle *)
		END_IF
	END_IF


5:	(* Release Node Handle *)
	fbUA_NodeReleaseHandle(
		Execute			:= TRUE,
		ConnectionHdl	:= nConnectionHdl,
		NodeHdl			:= nNodeHdl
	);

	IF NOT fbUA_NodeReleaseHandle.Busy THEN
		fbUA_NodeReleaseHandle(Execute := FALSE);

		IF NOT fbUA_NodeReleaseHandle.Error THEN
			iState 		:= iState + 1;
		ELSE
			bError		:= TRUE;
			nErrorID	:= fbUA_NodeReleaseHandle.ErrorID;
			iState 		:= 6; (* idle *)
		END_IF
	END_IF


6:	(* close session *)
	fbUA_Disconnect(
		Execute			:= TRUE,
		ConnectionHdl	:= nConnectionHdl
	);

	IF NOT fbUA_Disconnect.Busy THEN
		fbUA_Disconnect(Execute := FALSE);
		bBusy := FALSE; 
		IF NOT fbUA_Disconnect.Error THEN
			(* session closed *)
			iState 		:= 0;
			IF NOT bError THEN 
				bDone 	:= TRUE;
			END_IF
		ELSE
			bError			:= TRUE;
			nErrorID		:= fbUA_Disconnect.ErrorID;
			iState 			:= 0; (* idle *)
			nConnectionHdl	:= 0;
		END_IF
	END_IF
END_CASE

END_PROGRAM

// ---- POUs/PRG_WRITE_IndexRange.TcPOU
PROGRAM PRG_WRITE_IndexRange
VAR
	(* Declarations for UA_Connect *)
	fbUA_Connect			: UA_Connect;
	SessionConnectInfo		: ST_UASessionConnectInfo;
	nConnectionHdl			: DWORD;

	(* Declarations for UA_GetNamespaceIndex *)
	fbUA_GetNamespaceIndex 	: UA_GetNamespaceIndex;
	nNamespaceIndex			: UINT;

	(* Declarations for UA_NodeGetHandle *)
	fbUA_NodeGetHandle		: UA_NodeGetHandle;
	NodeID					: ST_UANodeID;
	nNodeHdl				: DWORD;

	(* Declarations for UA_Write *)
	fbUA_Write				: UA_Write;
	stIndexRange			: ARRAY [1..nMaxIndexRange] OF ST_UAIndexRange;
	nIndexRangeCount		: UINT;
	stNodeAddInfo			: ST_UANodeAdditionalInfo;
	sNodeIdentifier			: STRING(MAX_STRING_LENGTH) := '"IDB_Arrays_Typesafe"."MyDIntArray_Input"'; // change to node identifier
	nWriteData				: ARRAY[0..3] OF DINT;		// change according to the type of variable that should be written
	
	(* Declarations for UA_NodeReleaseHandle *)
	fbUA_NodeReleaseHandle	: UA_NodeReleaseHandle;

	(* Declarations for UA_Disconnect *)
	fbUA_Disconnect			: UA_Disconnect;

	(* Other declarations *)
	iState			: INT;
	bTest			: BOOL := TRUE;
	bDone			: BOOL;
	bBusy			: BOOL;
	bError			: BOOL;
	nErrorID		: DWORD;
END_VAR

CASE iState OF
0:	(* idle *)
	IF bTest THEN
		bTest	:= FALSE;
		bError	:= FALSE;
		nErrorID	:= 0;

		nWriteData[0] := 42;
		nWriteData[1] := 42;
		nWriteData[2] := 42;
		nWriteData[3] := 42;
		
		SessionConnectInfo.tConnectTimeout 		:= T#1M;
		SessionConnectInfo.tSessionTimeout 		:= T#1M;
		SessionConnectInfo.sApplicationName		:= '';
		SessionConnectInfo.eSecurityMode 		:= eUASecurityMsgMode_None;
		SessionConnectInfo.eSecurityPolicyUri 	:= eUASecurityPolicy_None;
		SessionConnectInfo.eTransportProfileUri := eUATransportProfileUri_UATcp;

		stIndexRange[1].nStartIndex := 2;
		stIndexRange[1].nEndIndex := 5;
		stNodeAddInfo.nIndexRangeCount := 1;
		stNodeAddInfo.stIndexRange := stIndexRange;
		
		iState	:= iState + 1;
	END_IF

1:	(* open UA session *)
	fbUA_Connect(
		Execute				:= TRUE,
		ServerURL			:= sOpcUaServerUrl,
		SessionConnectInfo	:= SessionConnectInfo,
		Timeout				:= T#2M,
		ConnectionHdl		=> nConnectionHdl
	);

	IF NOT fbUA_Connect.Busy THEN
		fbUA_Connect(Execute := FALSE);

		IF NOT fbUA_Connect.Error THEN
			(* session open *)
			iState := iState + 1;
		ELSE
			bError			:= TRUE;
			nErrorID		:= fbUA_Connect.ErrorID;
			nConnectionHdl	:= 0;
			iState 			:= 0; (* idle *)
		END_IF
	END_IF


2:	(* GetNS Index *)
	fbUA_GetNamespaceIndex(
		Execute			:= TRUE,
		ConnectionHdl	:= nConnectionHdl,
		NamespaceUri	:= sNamespaceUri,
		NamespaceIndex	=> nNamespaceIndex
	);

	IF NOT fbUA_GetNamespaceIndex.Busy THEN
		fbUA_GetNamespaceIndex(Execute := FALSE);

		IF NOT fbUA_GetNamespaceIndex.Error THEN
			iState 		:= iState + 1;
		ELSE
			bError		:= TRUE;
			nErrorID	:= fbUA_GetNamespaceIndex.ErrorID;
			iState 		:= 6; (* idle *)
		END_IF
	END_IF


3:	(* Get Node Handle *)
	NodeID.eIdentifierType := eUAIdentifierType_String;
	NodeID.nNamespaceIndex := nNamespaceIndex;
	NodeID.sIdentifier	:= sNodeIdentifier;
	fbUA_NodeGetHandle(
		Execute			:= TRUE,
		ConnectionHdl	:= nConnectionHdl,
		NodeID			:= NodeID,
		NodeHdl			=> nNodeHdl
	);

	IF NOT fbUA_NodeGetHandle.Busy THEN
		fbUA_NodeGetHandle(Execute := FALSE);

		IF NOT fbUA_NodeGetHandle.Error THEN
			iState 		:= iState + 1;
		ELSE
			bError		:= TRUE;
			nErrorID	:= fbUA_NodeGetHandle.ErrorID;
			iState 		:= 6; (* idle *)
		END_IF
	END_IF


4: 	(* UA_Write *)
	fbUA_Write(
		Execute			:= TRUE,
		ConnectionHdl	:= nConnectionHdl,
		NodeHdl			:= nNodeHdl,
		stNodeAddInfo	:= stNodeAddInfo,
		cbData			:= SIZEOF(nWriteData),
		pVariable		:= ADR(nWriteData)
		);

	IF NOT fbUA_Write.Busy THEN
		fbUA_Write(
			Execute 	:= FALSE,
			pVariable	:= ADR(nWriteData));

		IF NOT fbUA_Write.Error THEN
			iState 		:= iState + 1;
		ELSE
			bError		:= TRUE;
			nErrorID	:= fbUA_Write.ErrorID;
			iState 		:= 6; (* idle *)
		END_IF
	END_IF


5:	(* Release Node Handle *)
	fbUA_NodeReleaseHandle(
		Execute			:= TRUE,
		ConnectionHdl	:= nConnectionHdl,
		NodeHdl			:= nNodeHdl
	);

	IF NOT fbUA_NodeReleaseHandle.Busy THEN
		fbUA_NodeReleaseHandle(Execute := FALSE);

		IF NOT fbUA_NodeReleaseHandle.Error THEN
			iState 		:= iState + 1;
		ELSE
			bError		:= TRUE;
			nErrorID	:= fbUA_NodeReleaseHandle.ErrorID;
			iState 		:= 6; (* idle *)
		END_IF
	END_IF


6:	(* close session *)
	fbUA_Disconnect(
		Execute			:= TRUE,
		ConnectionHdl	:= nConnectionHdl
	);

	IF NOT fbUA_Disconnect.Busy THEN
		fbUA_Disconnect(Execute := FALSE);
		bBusy := FALSE; 
		IF NOT fbUA_Disconnect.Error THEN
			(* session closed *)
			iState 		:= 0;
			IF NOT bError THEN 
				bDone 	:= TRUE;
			END_IF
		ELSE
			bError			:= TRUE;
			nErrorID		:= fbUA_Disconnect.ErrorID;
			iState 			:= 0; (* idle *)
			nConnectionHdl	:= 0;
		END_IF
	END_IF
END_CASE

END_PROGRAM
